FUNCTION_BLOCK logiBUS_LED_strip_QX (* Output service interface function block for boolean output data *)
  (* Description: Copyright (c) 2014, 2015 fortiss GmbH This program and the accompanying materials are made available under the terms of the Eclipse Public License 2.0 which is available at https://www.eclipse.org/legal/epl-2.0/ SPDX-License-Identifier: EPL-2.0 *)
  (* Version 1.0, 2014-08-26, Waldemar Eisenmenger, fortiss GmbH *)
  (* Version 1.1, 2014-08-30, Alois Zoitl, fortiss GmbH *)
  (* Version 1.2, 2015-06-10, Monika Wenger, fortiss GmbH *)
  PACKAGE logiBUS::io::DO_LED;
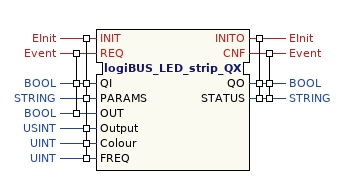
  EVENT_INPUT
    INIT : EInit WITH QI, PARAMS, Output, Colour, FREQ; (* Service Initialization *)
    REQ WITH QI, OUT; (* Service Request *)
  END_EVENT
  EVENT_OUTPUT
    INITO : EInit WITH QO, STATUS; (* Initialization Confirm *)
    CNF WITH QO, STATUS; (* Confirmation of Requested Service *)
  END_EVENT
  VAR_INPUT
    QI : BOOL; (* Event Input Qualifier *)
    PARAMS : STRING; (* Service Parameters *)
    OUT : BOOL; (* Output data to resource *)
    Output : USINT := LED_strip::Output_strip; (* Identify the Output Number of Strip *)
    Colour : UINT := LED_COLOURS::LED_GREEN; (* This identify the Colour. *)
    FREQ : UINT := LED_FREQ::LED_OFF; (* Define the LED Frequency and Priority *)
  END_VAR
  VAR_OUTPUT
    QO : BOOL; (* Event Output Qualifier *)
    STATUS : STRING; (* Service Status *)
  END_VAR
END_FUNCTION_BLOCK
